// TIA Portal V19 export
TYPE "PII - BCI24-DH367-1D1A-4"
   STRUCT
      "Process Data In - Switching output 1" : Bool;
      "Reserved Bit" : Bool;
      "Reserved Bit_1" : Bool;
      "Reserved Bit_2" : Bool;
      "Reserved Bit_3" : Bool;
      "Reserved Bit_4" : Bool;
      "Reserved Bit_5" : Bool;
      "Reserved Bit_6" : Bool;
      "Reserved Byte" : Bool;
      "Process Data In - Pressure" : Word;
      "Reserved Byte_1" : Bool;
      "Reserved Byte_2" : Bool;
      "Reserved Byte_3" : Bool;
      "Reserved Byte_4" : Bool;
      "Reserved Byte_5" : Bool;
      "Reserved Byte_6" : Bool;
      "Reserved Byte_7" : Bool;
      "Reserved Byte_8" : Bool;
      "Reserved Byte_9" : Bool;
      "Reserved Byte_10" : Bool;
      "Reserved Byte_11" : Bool;
      "Reserved Byte_12" : Bool;
      "Reserved Byte_13" : Bool;
      "Reserved Byte_14" : Bool;
      "Reserved Byte_15" : Bool;
      "Reserved Byte_16" : Bool;
      "Reserved Byte_17" : Bool;
      "Reserved Byte_18" : Bool;
      "Reserved Byte_19" : Bool;
      "Reserved Byte_20" : Bool;
      "Reserved Byte_21" : Bool;
      "Reserved Byte_22" : Bool;
      "Reserved Byte_23" : Bool;
      "Reserved Byte_24" : Bool;
      "Reserved Byte_25" : Bool;
      "Reserved Byte_26" : Bool;
      "Reserved Byte_27" : Bool;
      "Reserved Byte_28" : Bool;
      "Port qualifier" : Byte;
   END_STRUCT;
END_TYPE
